(*
SPDX-FileCopyrightText: © 2026 Oleksandr Tiutyk <trofimich@gmail.com>
SPDX-License-Identifier: MIT
License: https://opensource.org/license/mit
*)

INTERFACE ICompositeCondition EXTENDS ICondition

METHOD AddChildCondition
VAR_INPUT
	condition : ICondition;
END_VAR
END_METHOD

PROPERTY LogicalOperator : LOGICAL_OPERATOR
GET
END_GET
SET
END_SET
END_PROPERTY

END_INTERFACE

(* stored: Version 1.1.0.1
   Itf ICompositeCondition: Id {5071de02-a2b1-4cba-93bf-27c0973efb35}
   Method AddChildCondition: Id {dc921a49-202f-47b9-adb5-2f8dad5d5097}
   Property LogicalOperator: Id {30ffe6f4-aae4-4362-aacc-960e71565572}
   Get Get: Id {e3fc3c86-048d-4ff0-a309-84663d1eab60}
   Set Set: Id {f9275521-91e9-460d-b8b6-72fa668ebc4c} *)
